(* Logix 5000 project; controller StartingFile_DamonPark vendor 1 type 14 code 106 rev 28.11; software revision 28.03 *)

TASK MainTask (continuous, watchdog 500 ms) : MainProgram

MODULES
   Local : vendor 1 type 14 code 106 (Compact 0, rev 28.11)
       : 1769-IQ16 (Compact 3, rev 1.1, Input RPI 20 ms)
       : vendor 1 type 7 code 77 (Compact 2, rev 3.1, Input RPI 20 ms)
       : 1769-IF4 (Compact 6, rev 2.1, Input RPI 80 ms)
       : vendor 1 type 7 code 72 (Compact 4, rev 2.1, Output RPI 20 ms)
       : vendor 1 type 7 code 72 (Compact 5, rev 2.1, Output RPI 20 ms)
       : 1769-OF2 (Compact 7, rev 2.1, Output RPI 80 ms)
       : vendor 1 type 12 code 105 (Compact 1, rev 2.2, Output RPI 20 ms)
END_MODULES

TYPE DATETIME :
STRUCT
   Year : DINT;
   Month : DINT;
   Day : DINT;
   Hour : DINT;
   Minute : DINT;
   Second : DINT;
   Microseconds : DINT;
END_STRUCT
END_TYPE

TYPE StatAnalysis :
STRUCT
   F1_Call : DINT;
   F2_Call : DINT;
   F3_Call : DINT;
   F4_Call : DINT;
END_STRUCT
END_TYPE

VAR_GLOBAL   (* controller tags *)
   CR0 : ALIAS FOR Local:5:O.Data.4;   // Changes the direction of the M0
   Current_Floor : DINT := 1;   // Show which floor the elevator is located
   Current_State : DINT;   // Current State of the FSM
   D_Current_State : DINT;   // Current Door State of the Door State machine
   D_Next_State : DINT;   // Accepted Next Door State of the Door State machine
   DCLS : ALIAS FOR Local:3:I.Data.8;   // Door Close Limit Switch
   DOLS : ALIAS FOR Local:3:I.Data.9;   // Door Open Limit Switch
   Door_5s : TIMER := (PRE := 5000);   // 5 second timer Door closes 5sec after open
   Downmode : DINT;   // Saves the floor if the called floor is lower than current floor
   EMERGENCY : BOOL;   // True when the state is State_100_Emergency. Controls MCR
   Enable_PB : TIMER := (PRE := 2000);   // 2 second timer Enable the PBC 2 sec after door open
   F1 : DINT := 1;   // Floor1 = 1
   F2 : DINT := 2;   // Floor2 = 2
   F3 : DINT := 3;   // Floor3 = 3
   F4 : DINT := 4;   // Floor4 = 4
   FIL1 : ALIAS FOR Local:4:O.Data.11;   // Floor1 Indicator Light
   FIL2 : ALIAS FOR Local:4:O.Data.10;   // Floor2 Indicator Light
   FIL3 : ALIAS FOR Local:4:O.Data.9;   // Floor3 Indicator Light
   FIL4 : ALIAS FOR Local:4:O.Data.8;   // Floor4 Indicator Light
   FLS1 : ALIAS FOR Local:3:I.Data.0;   // Floor1 Limit Swtich
   FLS2 : ALIAS FOR Local:3:I.Data.1;   // Floor2 Indicator Light
   FLS3 : ALIAS FOR Local:3:I.Data.2;   // Floor3 Indicator Light
   FLS4 : ALIAS FOR Local:3:I.Data.3;   // Floor4 Indicator Light
   FPB1 : ALIAS FOR Local:2:I.Data.11;   // Floor1 Push Button
   FPB2 : ALIAS FOR Local:2:I.Data.10;   // Floor2 Indicator Light
   FPB3 : ALIAS FOR Local:2:I.Data.9;   // Floor3 Indicator Light
   FPB4 : ALIAS FOR Local:2:I.Data.8;   // Floor4 Indicator Light
   HMI_FPB1 : BOOL;
   HMI_FPB2 : BOOL;
   HMI_FPB3 : BOOL;
   HMI_FPB4 : BOOL;
   HMI_PB1 : BOOL;
   HMI_PB2 : BOOL;
   HMI_PB3 : BOOL;
   HMI_PB4 : BOOL;
   HMI_PBC : BOOL;
   HMI_PBE5 : BOOL;
   HMI_PBO : BOOL;
   IL1 : ALIAS FOR Local:4:O.Data.3;   // Indicator Light1
   IL2 : ALIAS FOR Local:4:O.Data.2;   // Indicator Light2
   IL3 : ALIAS FOR Local:4:O.Data.1;
   IL4 : ALIAS FOR Local:4:O.Data.0;
   ILC : ALIAS FOR Local:4:O.Data.5;
   ILE5 : ALIAS FOR Local:4:O.Data.6;
   ILO : ALIAS FOR Local:4:O.Data.4;
   ILTS0 : ALIAS FOR Local:4:O.Data.14;   // Indicator Light Toggle Switch 0
   ILTS1 : ALIAS FOR Local:4:O.Data.13;   // Indicator Light Toggle SW1
   ILTS2 : ALIAS FOR Local:4:O.Data.12;
   M0 : ALIAS FOR Local:5:O.Data.0;
   MCPV_A : ALIAS FOR Local:5:O.Data.13;
   MCPV_B : ALIAS FOR Local:5:O.Data.15;
   MCPV_EN : ALIAS FOR Local:5:O.Data.11;
   MCPV_FB : ALIAS FOR Local:3:I.Data.14;
   Next_State : DINT;   // Accepted Next Door State of the FSM
   ONS1 : BOOL;   // Oneshot 1
   ONS2 : BOOL;   // Oneshot 2
   ONS3 : BOOL;   // Oneshot 3
   ONS4 : BOOL;   // Oneshot 4
   ONS_F1 : BOOL;   // Oneshot for FLS1
   ONS_F2 : BOOL;   // Oneshot for FLS2
   ONS_F3 : BOOL;   // Oneshot for FLS3
   ONS_F4 : BOOL;   // Oneshot for FLS4
   OPEN_F1 : BOOL;   // True when (FPB1 or PB1) and FLS1
   OPEN_F2 : BOOL;   // True when (FPB2 or PB2) and FLS2
   OPEN_F3 : BOOL;   // True when (FPB3 or PB3) and FLS3
   OPEN_F4 : BOOL;   // True when (FPB4 or PB4) and FLS4
   PB1 : ALIAS FOR Local:2:I.Data.3;
   PB2 : ALIAS FOR Local:2:I.Data.2;
   PB3 : ALIAS FOR Local:2:I.Data.1;
   PB4 : ALIAS FOR Local:2:I.Data.0;
   PBC : ALIAS FOR Local:2:I.Data.5;
   PBE5 : ALIAS FOR Local:2:I.Data.6;
   PBO : ALIAS FOR Local:2:I.Data.4;
   Prev_State : DINT := 90;   // Save the previous state that was in motion
   SOL0 : ALIAS FOR Local:5:O.Data.2;
   START : ALIAS FOR Local:2:I.Data.14;
   State_0_DC : DINT;   // Door closed state
   State_0_Idle : DINT;   // Wait until any of floor is called
   State_1000_btwFloor : DINT := 1000;   // Leave the door closed if the elevator is stopped in between floors in Emergency
   State_100_atFloor : DINT := 100;   // Door open if the elevator is stopped at floor in Emergency
   State_100_Emergency : DINT := 100;   // Stop the operation of the elevator
   State_1_DO : DINT := 1;   // Door Opened state
   State_1_F1 : DINT := 1;   // Move the Elevator to first floor once run or pressing START in Emergency
   State_90_UPmode : DINT := 90;   // Move the Elevator upward
   State_91_DOWNmode : DINT := 91;   // Move the Elevator downward
   State_99_Service : DINT := 99;   // Stop the Elevator at the floor and wait for the service
   STOP : ALIAS FOR Local:2:I.Data.15;
   TS0 : ALIAS FOR Local:3:I.Data.12;   // toggle switch 0
   TS1 : ALIAS FOR Local:3:I.Data.11;   // Toggle SW1
   TS2 : ALIAS FOR Local:3:I.Data.10;
   Upmode : DINT;   // Saves the floor if the called floor is higher than current floor
   V_CR0 : BOOL;   // Virtual Control Relay 0
   V_DCLS : BOOL := 1;   // Virtual Door Close Limit Switch
   V_DOLS : BOOL;   // Virtual Door Open Limit Switch
   V_FIL1 : BOOL;   // Virtual Floor Indicator Light 1
   V_FIL2 : BOOL;   // Virtual Floor Indicator Light 2
   V_FIL3 : BOOL;   // Virtual Floor Indicator Light 3
   V_FIL4 : BOOL;   // Virtual Floor Indicator Light 4
   V_FLS1 : BOOL := 1;   // Virtual Floor Limit Switch 1
   V_FLS2 : BOOL;   // Virtual Floor Limit Switch 2
   V_FLS3 : BOOL;   // Virtual Floor Limit Switch 3
   V_FLS4 : BOOL;   // Virtual Floor Limit Switch 4
   V_FPB1 : BOOL;   // Virtual Floor Pushbutton 1
   V_FPB2 : BOOL;   // Virtual Floor Pushbutton 2
   V_FPB3 : BOOL;   // Virtual Floor Pushbutton 3
   V_FPB4 : BOOL;   // Virtual Floor Pushbutton 4
   V_IL1 : BOOL;   // Virtual Indicator Light 1
   V_IL2 : BOOL;   // Virtual Indicator Light 2
   V_IL3 : BOOL;   // Virtual Indicator Light 3
   V_IL4 : BOOL;   // Virtual Indicator Light 4
   V_ILC : BOOL;   // Virtual Indicator Light Close
   V_ILE5 : BOOL;   // Virtual Indicator Light Emergency 5
   V_ILO : BOOL;   // Virtual Indicator Light Open
   V_ILTS0 : BOOL;   // Vitual Indicator Light Toggle Switch 0
   V_ILTS1 : BOOL;   // Virtual Indicator Light Toggle Switch 1
   V_ILTS2 : BOOL;   // Virtual Indicator Light Toggle Switch 2
   V_M0 : BOOL;   // Virtual Motor 0
   V_PB1 : BOOL;   // Virtual Pushbutton 1
   V_PB2 : BOOL;   // Virtual Pushbutton 2
   V_PB3 : BOOL;   // Virtual Pushbutton 3
   V_PB4 : BOOL;   // Virtual Pushbutton 4
   V_PBC : BOOL;   // Virtual Pushbutton Close
   V_PBE5 : BOOL;   // Virtual Pushbutton Emergency 5
   V_PBO : BOOL;   // Virtual Pushbutton Open
   V_SOL0 : BOOL;   // Virtual Solenoid 0
   V_START : BOOL;   // Virtual Start Button (N.O.)
   V_STOP : BOOL := 1;   // Virtual Stop Button (N.C.)
   V_TS0 : BOOL;   // Virtual Toggle Switch 0
   V_TS1 : BOOL;   // Virtual Toggle Switch 1
   V_TS2 : BOOL;   // Virtual Toggle Switch 2
END_VAR

PROGRAM MainProgram   (* main routine MainRoutine *)

ROUTINE Buffer   (* ladder *)
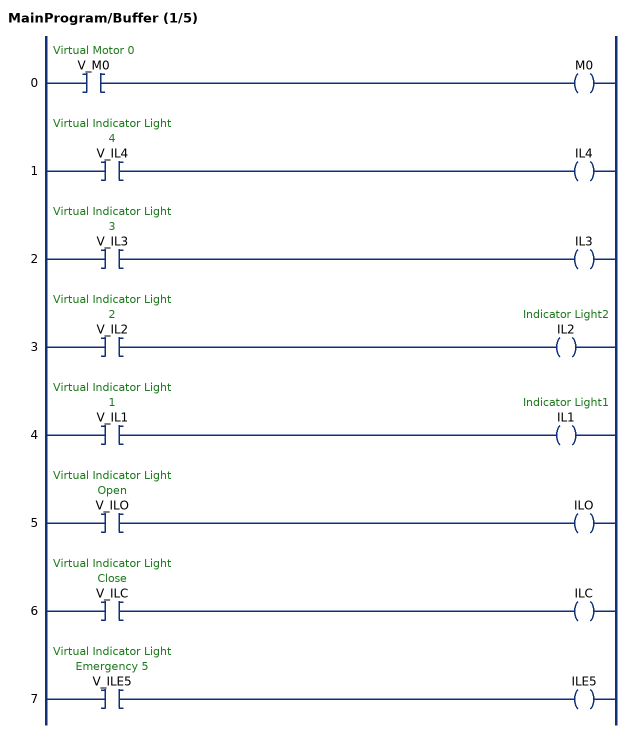
   0: XIC(V_M0)OTE(M0);
   1: XIC(V_IL4)OTE(IL4);
   2: XIC(V_IL3)OTE(IL3);
   3: XIC(V_IL2)OTE(IL2);
   4: XIC(V_IL1)OTE(IL1);
   5: XIC(V_ILO)OTE(ILO);
   6: XIC(V_ILC)OTE(ILC);
   7: XIC(V_ILE5)OTE(ILE5);
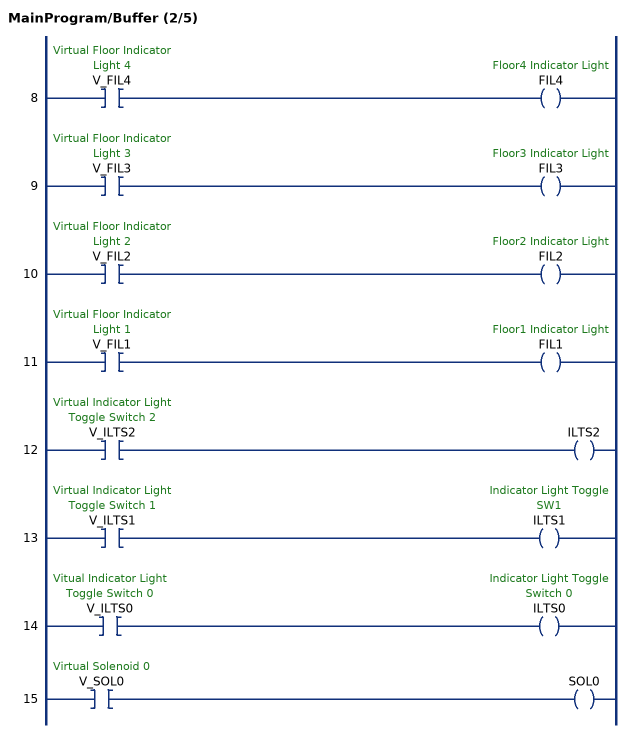
   8: XIC(V_FIL4)OTE(FIL4);
   9: XIC(V_FIL3)OTE(FIL3);
   10: XIC(V_FIL2)OTE(FIL2);
   11: XIC(V_FIL1)OTE(FIL1);
   12: XIC(V_ILTS2)OTE(ILTS2);
   13: XIC(V_ILTS1)OTE(ILTS1);
   14: XIC(V_ILTS0)OTE(ILTS0);
   15: XIC(V_SOL0)OTE(SOL0);
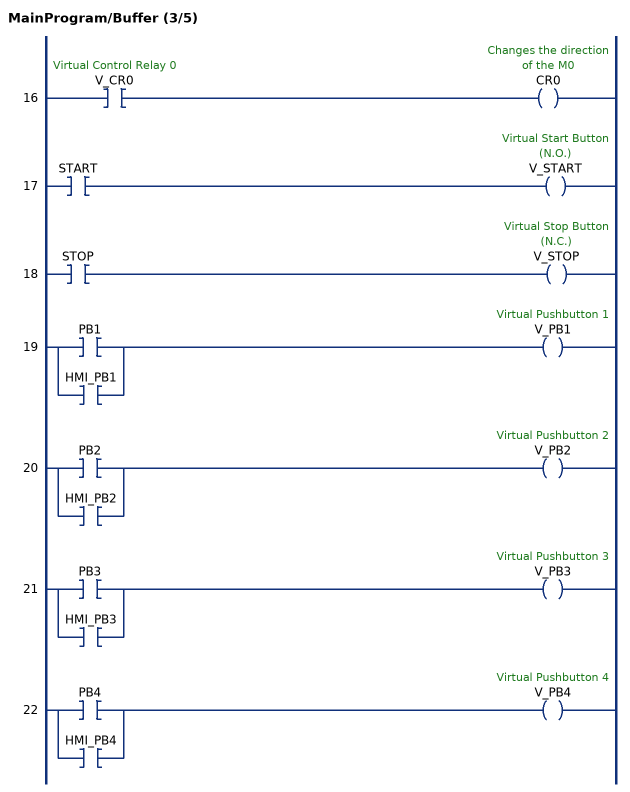
   16: XIC(V_CR0)OTE(CR0);
   17: XIC(START)OTE(V_START);
   18: XIC(STOP)OTE(V_STOP);
   19: [XIC(PB1) ,XIC(HMI_PB1) ]OTE(V_PB1);
   20: [XIC(PB2) ,XIC(HMI_PB2) ]OTE(V_PB2);
   21: [XIC(PB3) ,XIC(HMI_PB3) ]OTE(V_PB3);
   22: [XIC(PB4) ,XIC(HMI_PB4) ]OTE(V_PB4);
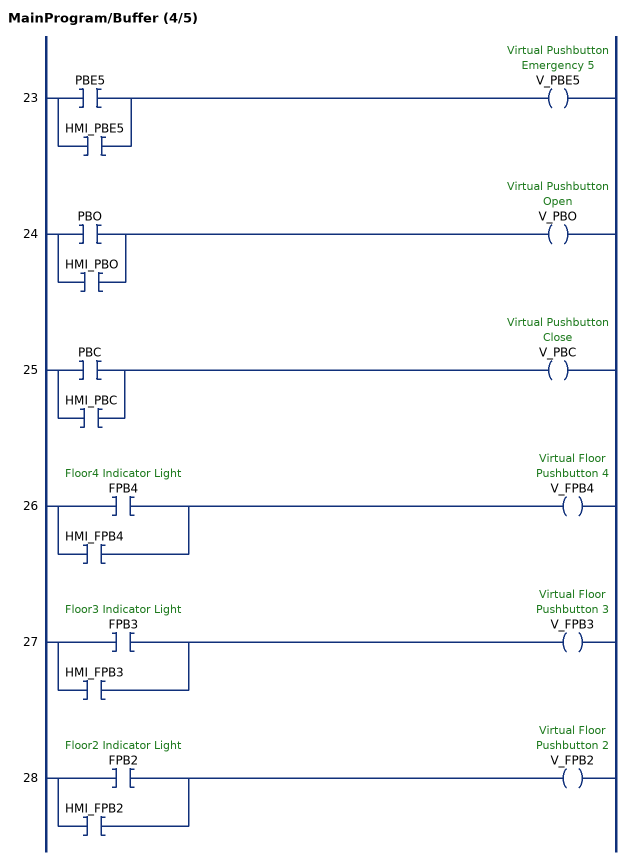
   23: [XIC(PBE5) ,XIC(HMI_PBE5) ]OTE(V_PBE5);
   24: [XIC(PBO) ,XIC(HMI_PBO) ]OTE(V_PBO);
   25: [XIC(PBC) ,XIC(HMI_PBC) ]OTE(V_PBC);
   26: [XIC(FPB4) ,XIC(HMI_FPB4) ]OTE(V_FPB4);
   27: [XIC(FPB3) ,XIC(HMI_FPB3) ]OTE(V_FPB3);
   28: [XIC(FPB2) ,XIC(HMI_FPB2) ]OTE(V_FPB2);
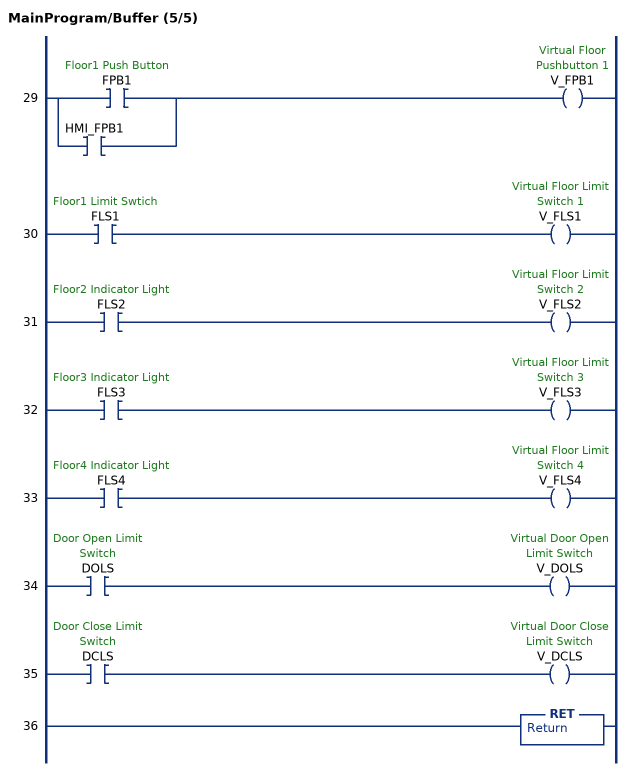
   29: [XIC(FPB1) ,XIC(HMI_FPB1) ]OTE(V_FPB1);
   30: XIC(FLS1)OTE(V_FLS1);
   31: XIC(FLS2)OTE(V_FLS2);
   32: XIC(FLS3)OTE(V_FLS3);
   33: XIC(FLS4)OTE(V_FLS4);
   34: XIC(DOLS)OTE(V_DOLS);
   35: XIC(DCLS)OTE(V_DCLS);
   36: RET();
END_ROUTINE

ROUTINE Door   (* ladder *)
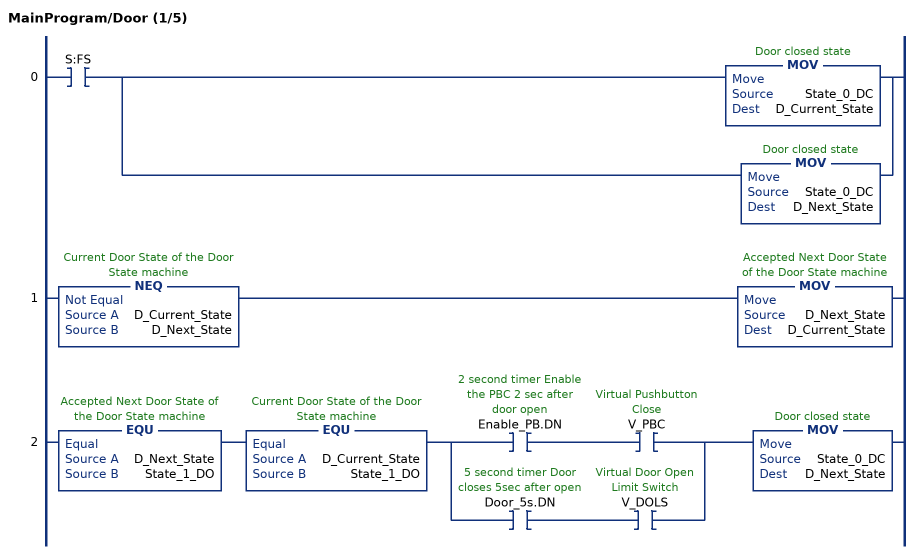
   0: XIC(S:FS)[MOV(State_0_DC,D_Current_State) ,MOV(State_0_DC,D_Next_State) ];
   1: NEQ(D_Current_State,D_Next_State)MOV(D_Next_State,D_Current_State);
   2: EQU(D_Next_State,State_1_DO)EQU(D_Current_State,State_1_DO)[XIC(Enable_PB.DN) XIC(V_PBC) ,XIC(Door_5s.DN) XIC(V_DOLS) ]MOV(State_0_DC,D_Next_State);
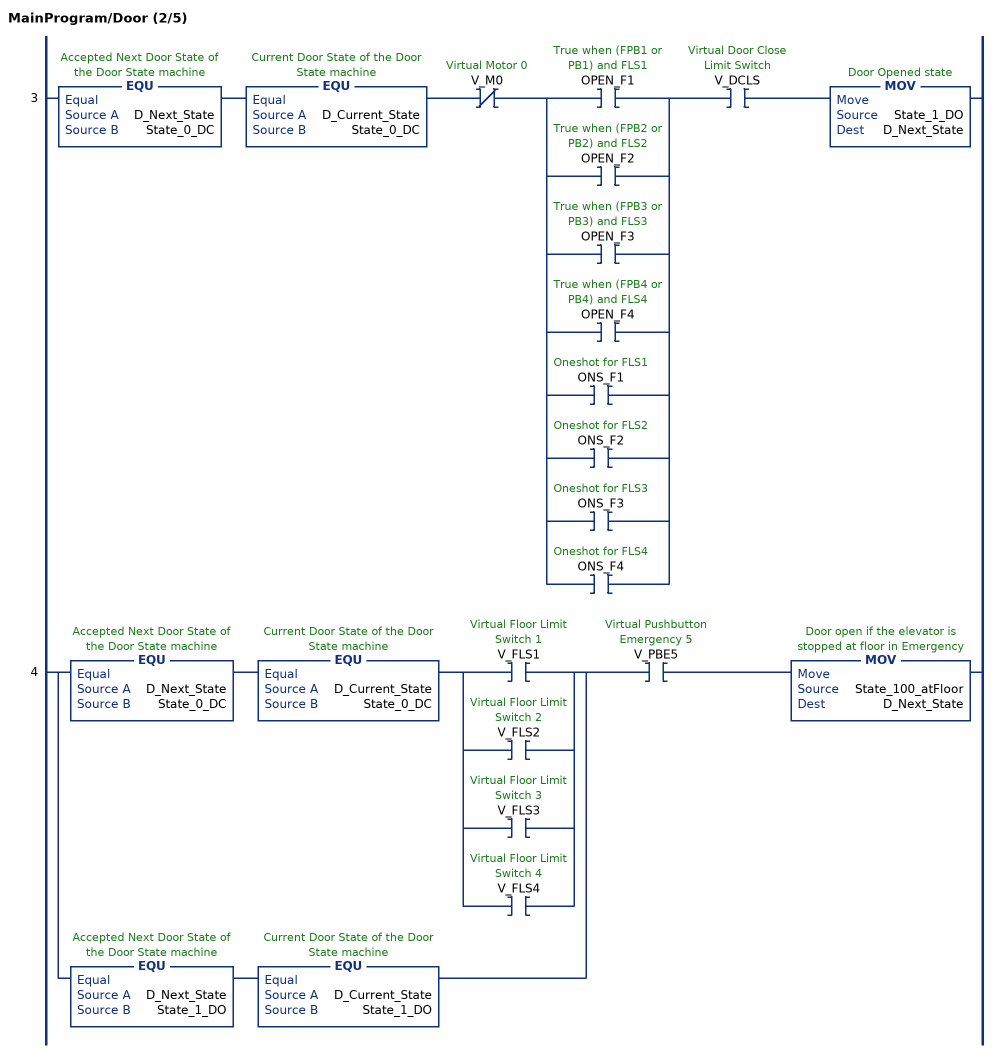
   3: EQU(D_Next_State,State_0_DC)EQU(D_Current_State,State_0_DC)XIO(V_M0)[XIC(OPEN_F1) ,XIC(OPEN_F2) ,XIC(OPEN_F3) ,XIC(OPEN_F4) ,XIC(ONS_F1) ,XIC(ONS_F2) ,XIC(ONS_F3) ,XIC(ONS_F4) ]XIC(V_DCLS)MOV(State_1_DO,D_Next_State);
   4: [EQU(D_Next_State,State_0_DC) EQU(D_Current_State,State_0_DC) [XIC(V_FLS1) ,XIC(V_FLS2) ,XIC(V_FLS3) ,XIC(V_FLS4) ] ,EQU(D_Next_State,State_1_DO) EQU(D_Current_State,State_1_DO) ]XIC(V_PBE5)MOV(State_100_atFloor,D_Next_State);
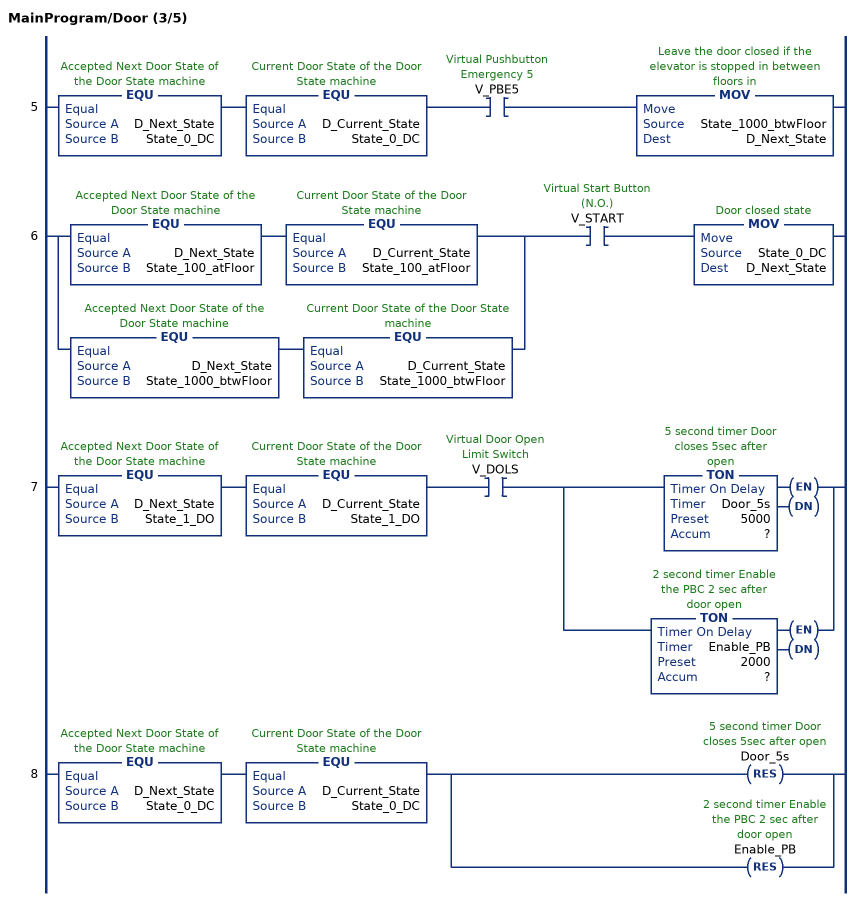
   5: EQU(D_Next_State,State_0_DC)EQU(D_Current_State,State_0_DC)XIC(V_PBE5)MOV(State_1000_btwFloor,D_Next_State);
   6: [EQU(D_Next_State,State_100_atFloor) EQU(D_Current_State,State_100_atFloor) ,EQU(D_Next_State,State_1000_btwFloor) EQU(D_Current_State,State_1000_btwFloor) ]XIC(V_START)MOV(State_0_DC,D_Next_State);
   7: EQU(D_Next_State,State_1_DO)EQU(D_Current_State,State_1_DO)XIC(V_DOLS)[TON(Door_5s,?,?) ,TON(Enable_PB,?,?) ];
   8: EQU(D_Next_State,State_0_DC)EQU(D_Current_State,State_0_DC)[RES(Door_5s) ,RES(Enable_PB) ];
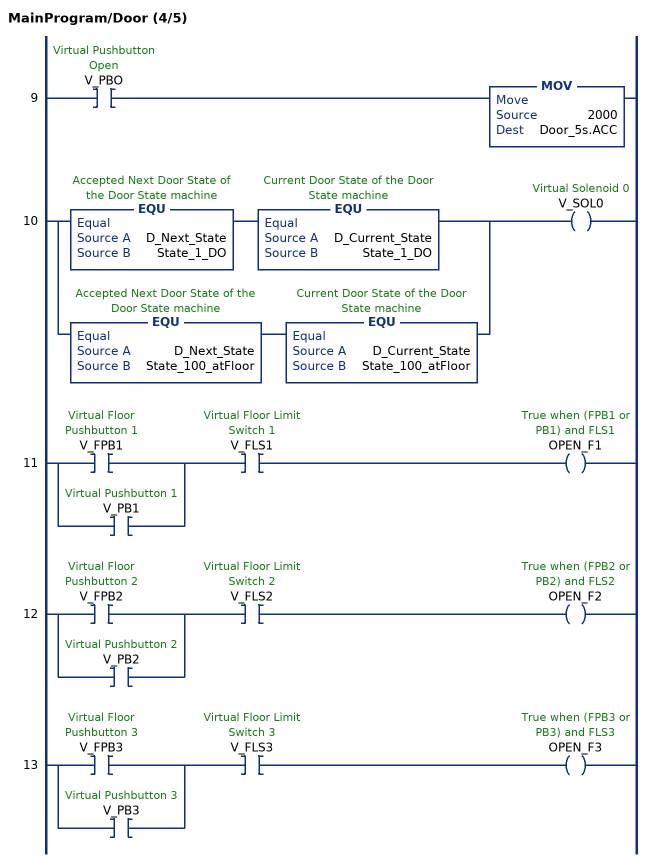
   9: XIC(V_PBO)MOV(2000,Door_5s.ACC);
   10: [EQU(D_Next_State,State_1_DO) EQU(D_Current_State,State_1_DO) ,EQU(D_Next_State,State_100_atFloor) EQU(D_Current_State,State_100_atFloor) ]OTE(V_SOL0);
   11: [XIC(V_FPB1) ,XIC(V_PB1) ]XIC(V_FLS1)OTE(OPEN_F1);
   12: [XIC(V_FPB2) ,XIC(V_PB2) ]XIC(V_FLS2)OTE(OPEN_F2);
   13: [XIC(V_FPB3) ,XIC(V_PB3) ]XIC(V_FLS3)OTE(OPEN_F3);
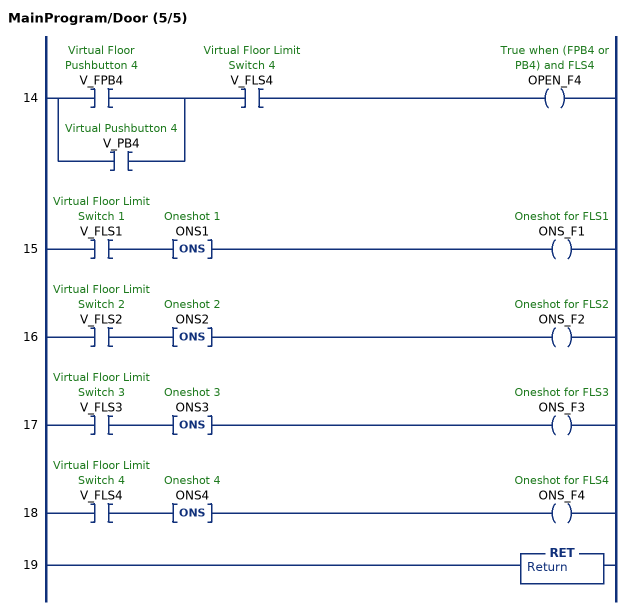
   14: [XIC(V_FPB4) ,XIC(V_PB4) ]XIC(V_FLS4)OTE(OPEN_F4);
   15: XIC(V_FLS1)ONS(ONS1)OTE(ONS_F1);
   16: XIC(V_FLS2)ONS(ONS2)OTE(ONS_F2);
   17: XIC(V_FLS3)ONS(ONS3)OTE(ONS_F3);
   18: XIC(V_FLS4)ONS(ONS4)OTE(ONS_F4);
   19: RET();
END_ROUTINE

ROUTINE Floorcall   (* ladder *)
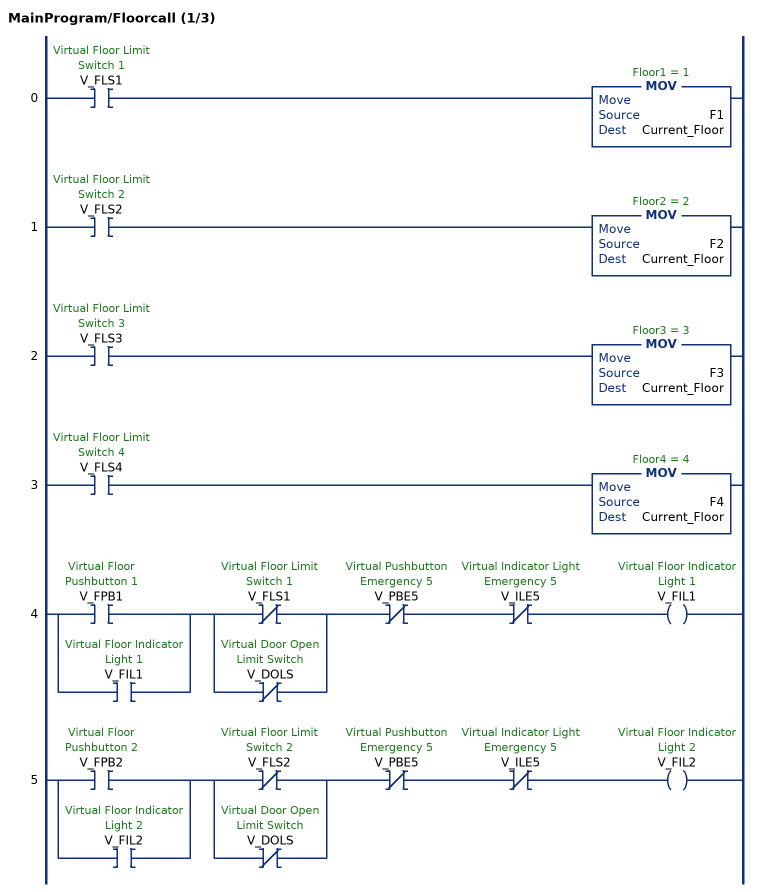
   0: XIC(V_FLS1)MOV(F1,Current_Floor);
   1: XIC(V_FLS2)MOV(F2,Current_Floor);
   2: XIC(V_FLS3)MOV(F3,Current_Floor);
   3: XIC(V_FLS4)MOV(F4,Current_Floor);
   4: [XIC(V_FPB1) ,XIC(V_FIL1) ][XIO(V_FLS1) ,XIO(V_DOLS) ]XIO(V_PBE5)XIO(V_ILE5)OTE(V_FIL1);
   5: [XIC(V_FPB2) ,XIC(V_FIL2) ][XIO(V_FLS2) ,XIO(V_DOLS) ]XIO(V_PBE5)XIO(V_ILE5)OTE(V_FIL2);
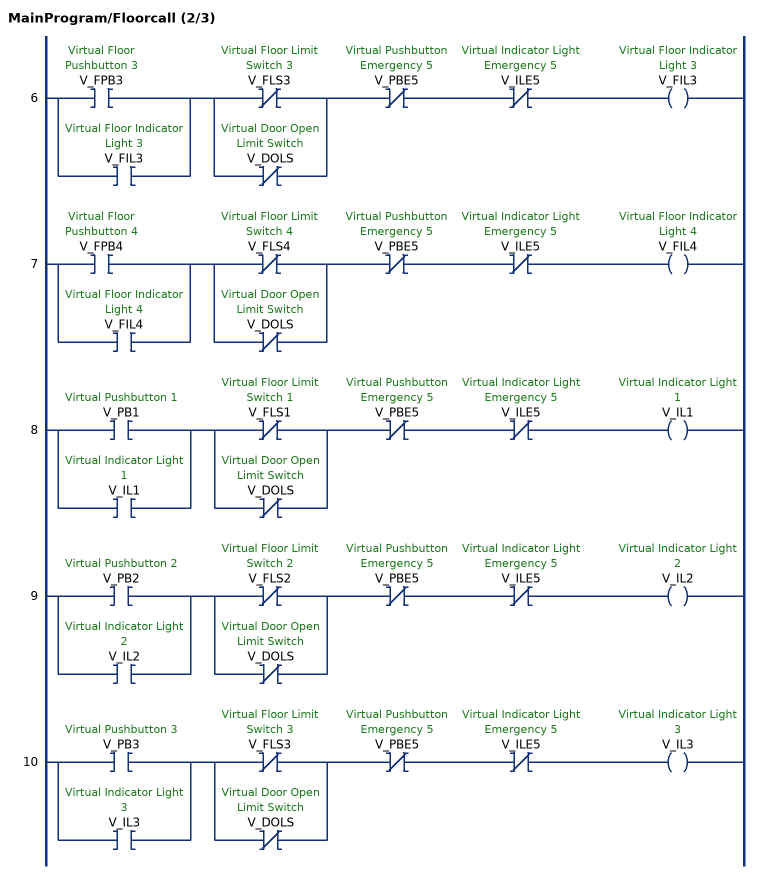
   6: [XIC(V_FPB3) ,XIC(V_FIL3) ][XIO(V_FLS3) ,XIO(V_DOLS) ]XIO(V_PBE5)XIO(V_ILE5)OTE(V_FIL3);
   7: [XIC(V_FPB4) ,XIC(V_FIL4) ][XIO(V_FLS4) ,XIO(V_DOLS) ]XIO(V_PBE5)XIO(V_ILE5)OTE(V_FIL4);
   8: [XIC(V_PB1) ,XIC(V_IL1) ][XIO(V_FLS1) ,XIO(V_DOLS) ]XIO(V_PBE5)XIO(V_ILE5)OTE(V_IL1);
   9: [XIC(V_PB2) ,XIC(V_IL2) ][XIO(V_FLS2) ,XIO(V_DOLS) ]XIO(V_PBE5)XIO(V_ILE5)OTE(V_IL2);
   10: [XIC(V_PB3) ,XIC(V_IL3) ][XIO(V_FLS3) ,XIO(V_DOLS) ]XIO(V_PBE5)XIO(V_ILE5)OTE(V_IL3);
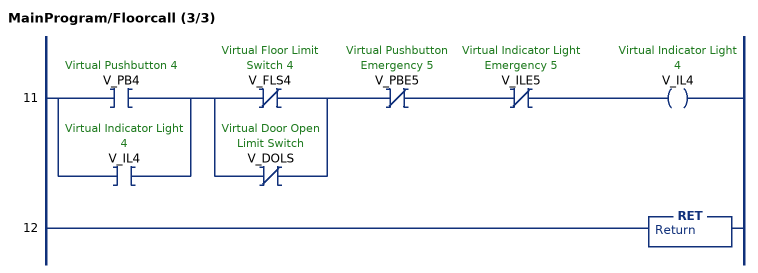
   11: [XIC(V_PB4) ,XIC(V_IL4) ][XIO(V_FLS4) ,XIO(V_DOLS) ]XIO(V_PBE5)XIO(V_ILE5)OTE(V_IL4);
   12: RET();
END_ROUTINE

ROUTINE MainRoutine   (* ladder *)
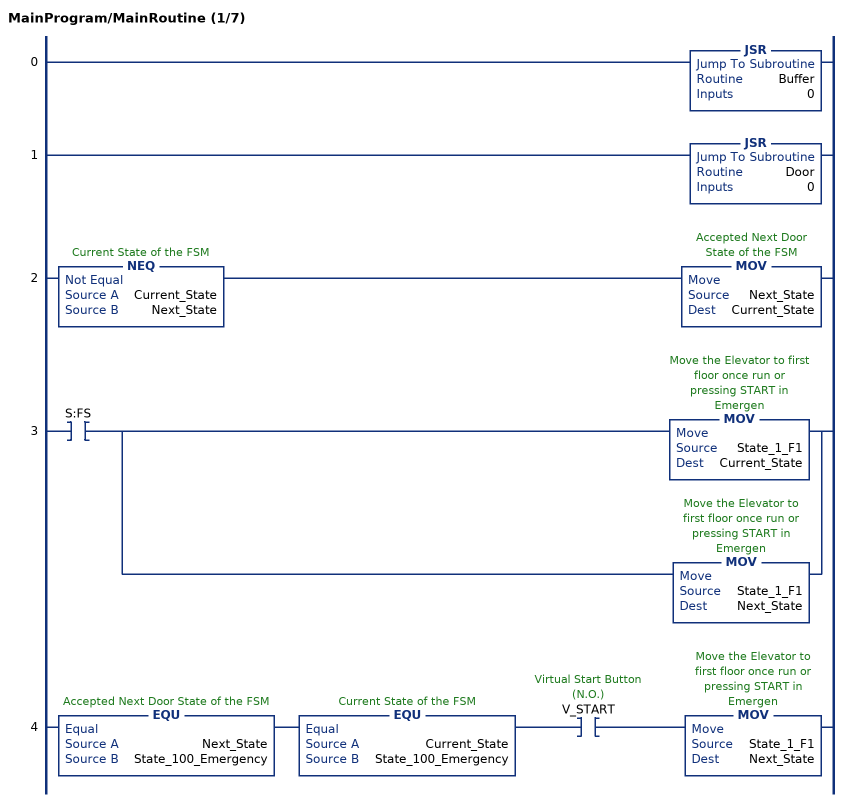
   0: JSR(Buffer,0);
   1: JSR(Door,0);
   2: NEQ(Current_State,Next_State)MOV(Next_State,Current_State);
   3: XIC(S:FS)[MOV(State_1_F1,Current_State) ,MOV(State_1_F1,Next_State) ];
   4: EQU(Next_State,State_100_Emergency)EQU(Current_State,State_100_Emergency)XIC(V_START)MOV(State_1_F1,Next_State);
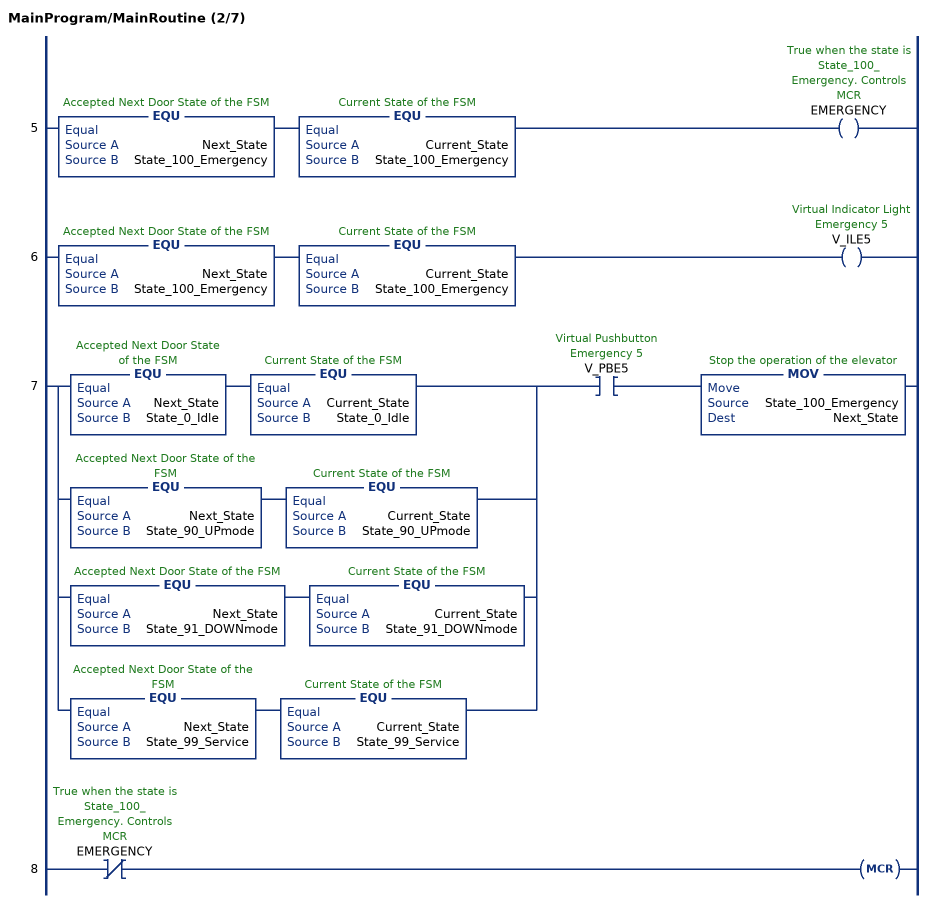
   5: EQU(Next_State,State_100_Emergency)EQU(Current_State,State_100_Emergency)OTE(EMERGENCY);
   6: EQU(Next_State,State_100_Emergency)EQU(Current_State,State_100_Emergency)OTE(V_ILE5);
   7: [EQU(Next_State,State_0_Idle) EQU(Current_State,State_0_Idle) ,EQU(Next_State,State_90_UPmode) EQU(Current_State,State_90_UPmode) ,[EQU(Next_State,State_91_DOWNmode) EQU(Current_State,State_91_DOWNmode) ,EQU(Next_State,State_99_Service) EQU(Current_State,State_99_Service) ] ]XIC(V_PBE5)MOV(State_100_Emergency,Next_State);
   8: XIO(EMERGENCY)MCR();
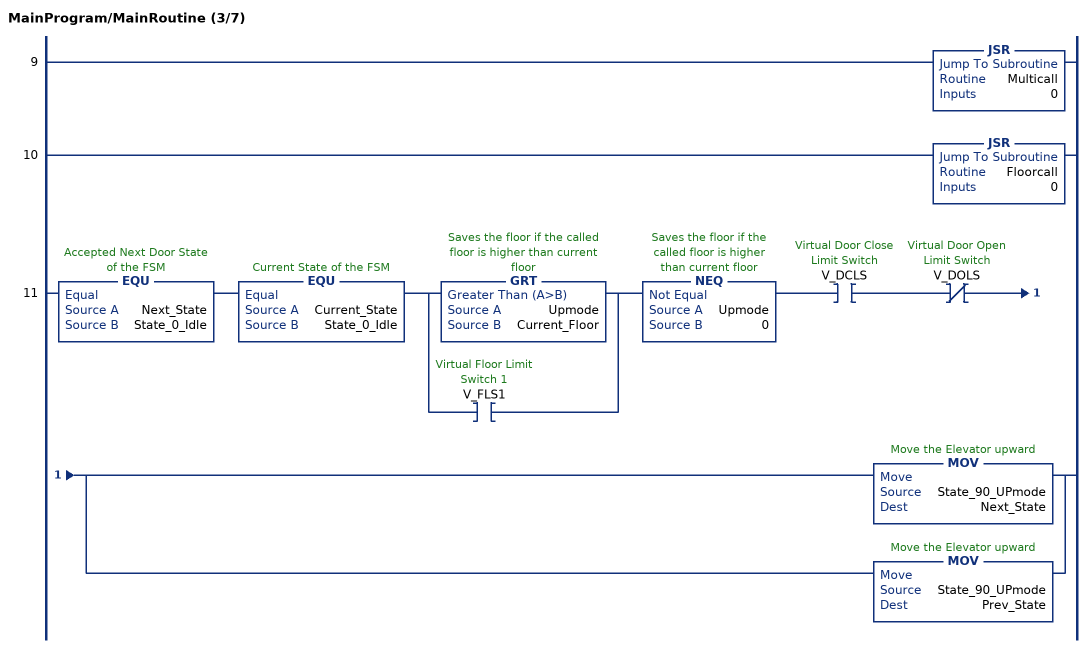
   9: JSR(Multicall,0);
   10: JSR(Floorcall,0);
   11: EQU(Next_State,State_0_Idle)EQU(Current_State,State_0_Idle)[GRT(Upmode,Current_Floor) ,XIC(V_FLS1) ]NEQ(Upmode,0)XIC(V_DCLS)XIO(V_DOLS)[MOV(State_90_UPmode,Next_State) ,MOV(State_90_UPmode,Prev_State) ];
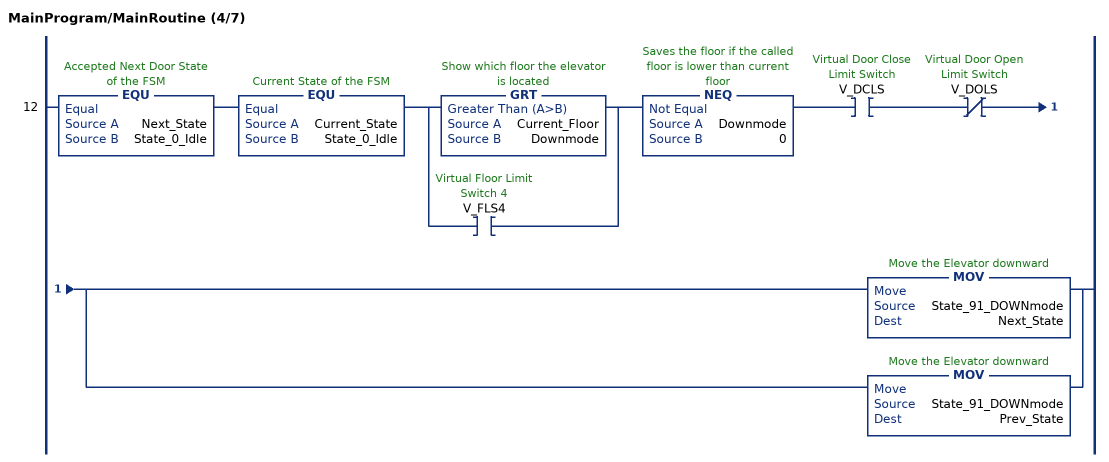
   12: EQU(Next_State,State_0_Idle)EQU(Current_State,State_0_Idle)[GRT(Current_Floor,Downmode) ,XIC(V_FLS4) ]NEQ(Downmode,0)XIC(V_DCLS)XIO(V_DOLS)[MOV(State_91_DOWNmode,Next_State) ,MOV(State_91_DOWNmode,Prev_State) ];
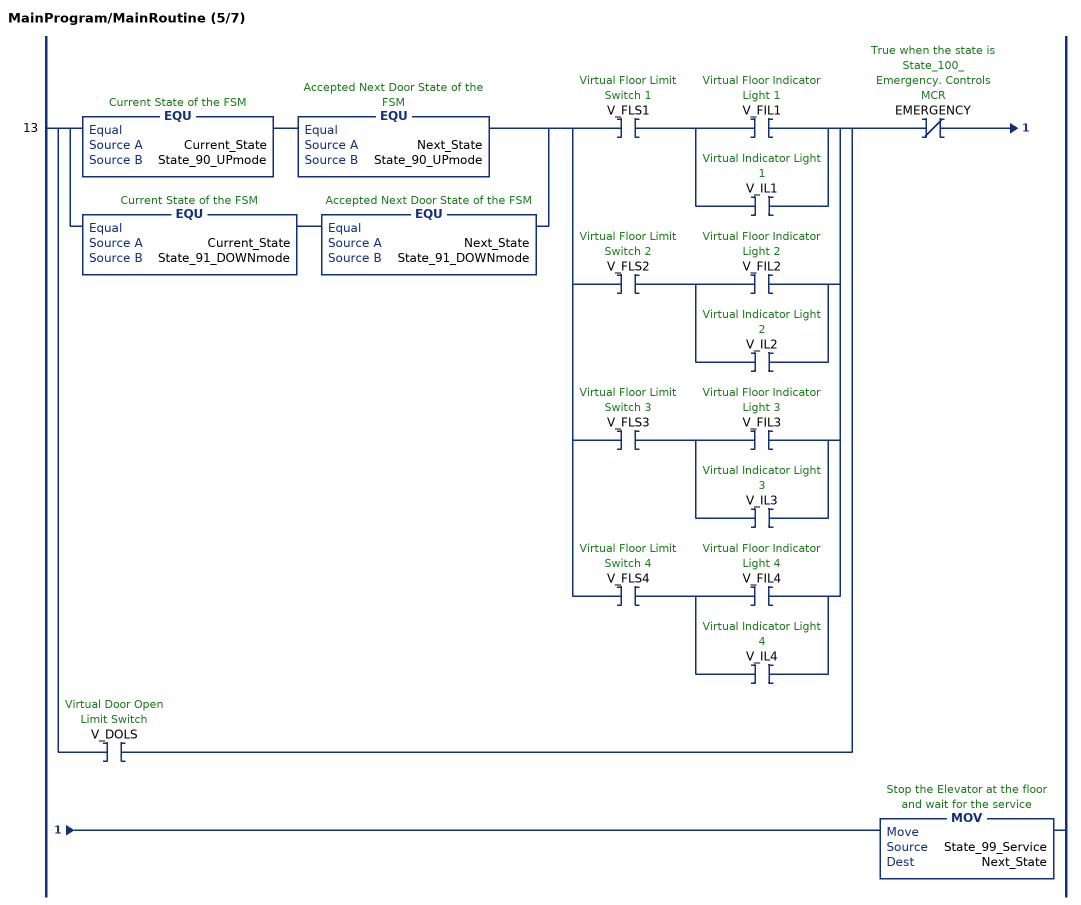
   13: [[EQU(Current_State,State_90_UPmode) EQU(Next_State,State_90_UPmode) ,EQU(Current_State,State_91_DOWNmode) EQU(Next_State,State_91_DOWNmode) ] [XIC(V_FLS1) [XIC(V_FIL1) ,XIC(V_IL1) ] ,XIC(V_FLS2) [XIC(V_FIL2) ,XIC(V_IL2) ] ,XIC(V_FLS3) [XIC(V_FIL3) ,XIC(V_IL3) ] ,XIC(V_FLS4) [XIC(V_FIL4) ,XIC(V_IL4) ] ] ,XIC(V_DOLS) ]XIO(EMERGENCY)MOV(State_99_Service,Next_State);
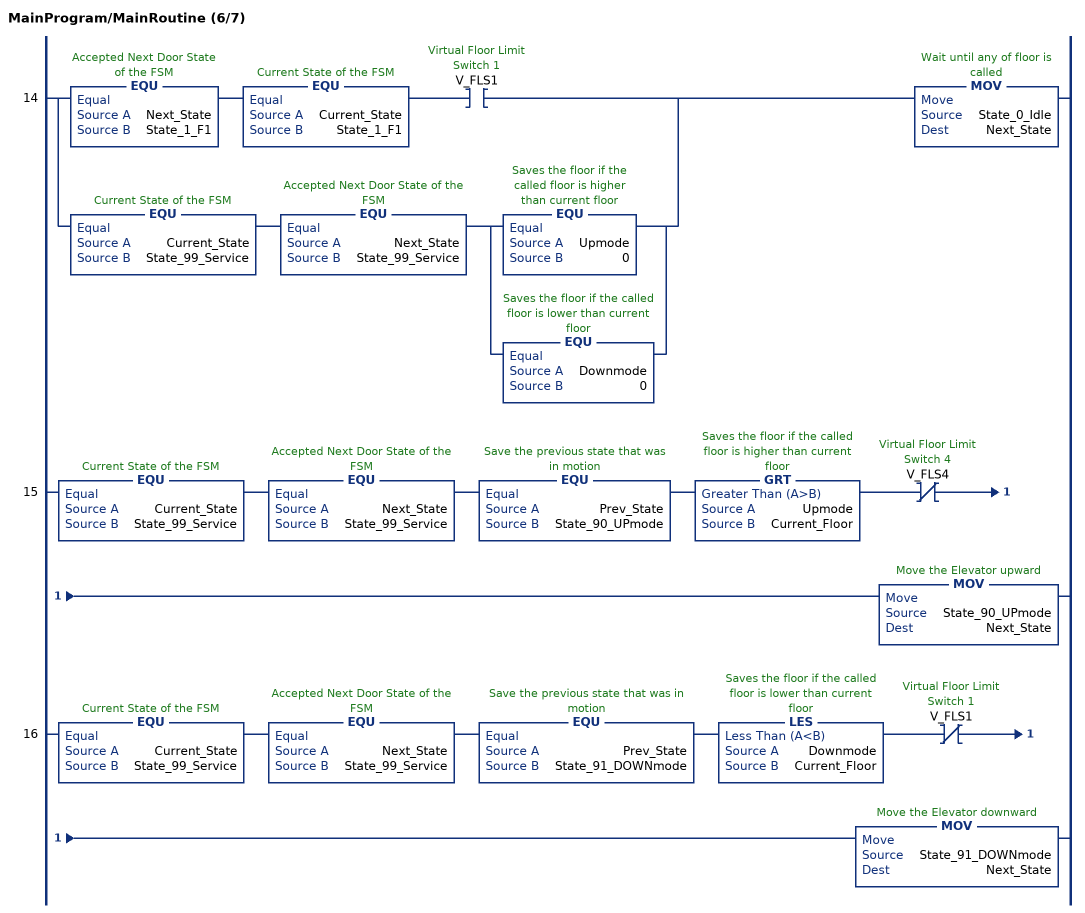
   14: [EQU(Next_State,State_1_F1) EQU(Current_State,State_1_F1) XIC(V_FLS1) ,EQU(Current_State,State_99_Service) EQU(Next_State,State_99_Service) [EQU(Upmode,0) ,EQU(Downmode,0) ] ]MOV(State_0_Idle,Next_State);
   15: EQU(Current_State,State_99_Service)EQU(Next_State,State_99_Service)EQU(Prev_State,State_90_UPmode)GRT(Upmode,Current_Floor)XIO(V_FLS4)MOV(State_90_UPmode,Next_State);
   16: EQU(Current_State,State_99_Service)EQU(Next_State,State_99_Service)EQU(Prev_State,State_91_DOWNmode)LES(Downmode,Current_Floor)XIO(V_FLS1)MOV(State_91_DOWNmode,Next_State);
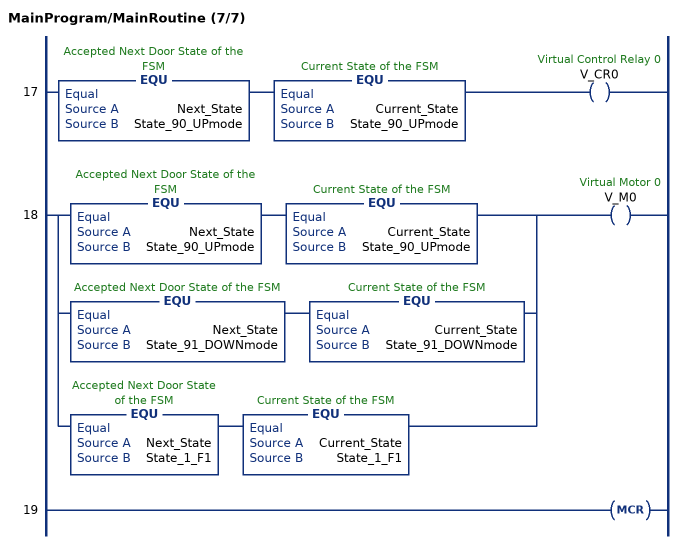
   17: EQU(Next_State,State_90_UPmode)EQU(Current_State,State_90_UPmode)OTE(V_CR0);
   18: [EQU(Next_State,State_90_UPmode) EQU(Current_State,State_90_UPmode) ,EQU(Next_State,State_91_DOWNmode) EQU(Current_State,State_91_DOWNmode) ,EQU(Next_State,State_1_F1) EQU(Current_State,State_1_F1) ]OTE(V_M0);
   19: MCR();
END_ROUTINE

ROUTINE Multicall   (* ladder *)
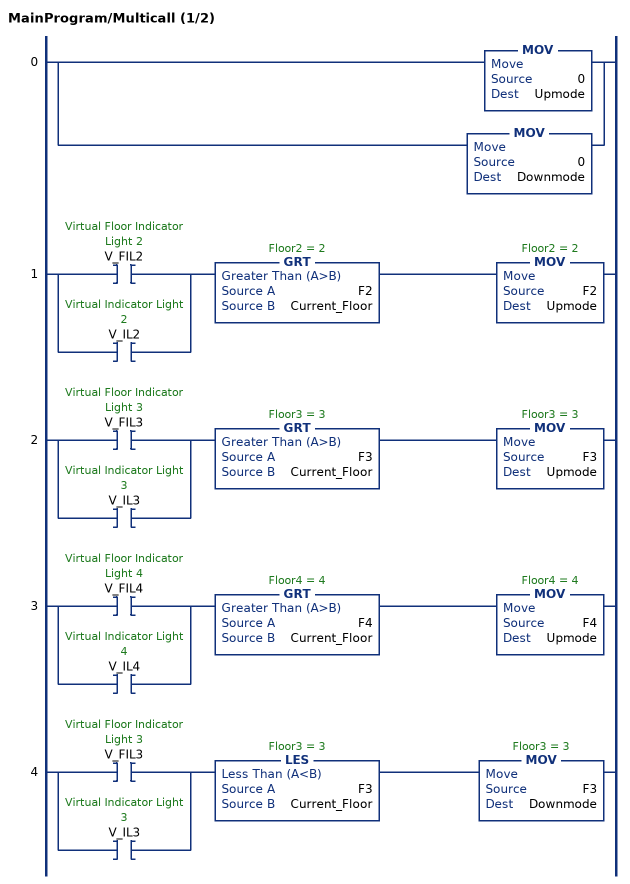
   0: [MOV(0,Upmode) ,MOV(0,Downmode) ];
   1: [XIC(V_FIL2) ,XIC(V_IL2) ]GRT(F2,Current_Floor)MOV(F2,Upmode);
   2: [XIC(V_FIL3) ,XIC(V_IL3) ]GRT(F3,Current_Floor)MOV(F3,Upmode);
   3: [XIC(V_FIL4) ,XIC(V_IL4) ]GRT(F4,Current_Floor)MOV(F4,Upmode);
   4: [XIC(V_FIL3) ,XIC(V_IL3) ]LES(F3,Current_Floor)MOV(F3,Downmode);
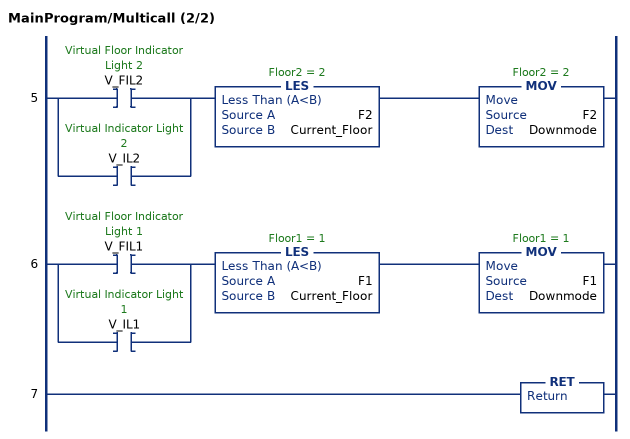
   5: [XIC(V_FIL2) ,XIC(V_IL2) ]LES(F2,Current_Floor)MOV(F2,Downmode);
   6: [XIC(V_FIL1) ,XIC(V_IL1) ]LES(F1,Current_Floor)MOV(F1,Downmode);
   7: RET();
END_ROUTINE
END_PROGRAM
